// TIA Portal project "Project4_V16" (V16)

(* hardware
DEVICE "S7-1200 station_2"  S7-1200 Station
   slot 0: "Rack_0"  S7-1200 Rack  Rack  V1.0
   slot 1: "PLC_TO_SCADA"  CPU 1214C DC/DC/DC  6ES7 214-1AG40-0XB0  V4.1
DEVICE "S7-1200 station_3"  S7-1200 Station
   slot 0: "Rack_0"  S7-1200 Rack  Rack  V1.0
   slot 1: "PLC_2"  CPU 1214C DC/DC/DC  6ES7 214-1AG40-0XB0  V4.1
DEVICE "S7-1200 station_1"  S7-1200 Station
   slot 0: "Rack_0"  S7-1200 Rack  Rack  V1.0
   slot 1: "PLC_1"  CPU 1212C DC/DC/Rly  6ES7 212-1HE40-0XB0  V4.2
*)

// ===== PLC "PLC_TO_SCADA"  CPU 1214C DC/DC/DC =====

VAR_GLOBAL   // PLC tag table "Default tag table"
   "Tag_1" AT %M0.0 : Bool;
   "Tag_2" AT %M0.1 : Bool;
   "Tag_3" AT %M0.5 : Bool;
   "Tag_4" AT %MD100 : Time;
   "Tag_5" AT %M0.2 : Bool;
   "Tag_6" AT %I0.0 : Bool;
   "Tag_7" AT %I0.1 : Bool;
END_VAR

// folder: System blocks/Program resources

DATA_BLOCK "t0"   // DB1
{ S7_Optimized_Access := 'TRUE' }
AUTHOR : Simatic
FAMILY : IEC
NAME : IEC_TMR
VERSION : 1.0
// stored: InstanceOfName IEC_TIMER
"IEC_TIMER"
BEGIN
END_DATA_BLOCK

// folder: (top level)

ORGANIZATION_BLOCK "Main"   // OB1, LAD, ProgramCycle
TITLE = "Main Program Sweep (Cycle)"
{ S7_Optimized_Access := 'TRUE' }
VERSION : 0.1
   VAR_INPUT
      Initial_Call : Bool;   // Initial call of this OB
      Remanence : Bool;   // =True, if remanent data are available
   END_VAR
BEGIN

REGION Network 1
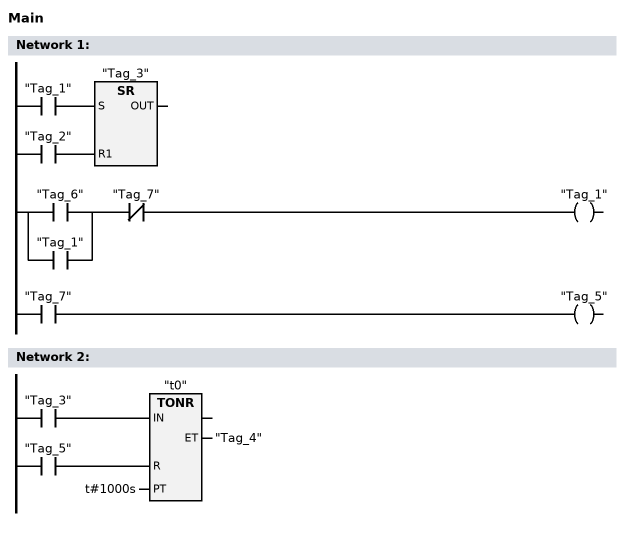
   RUNG wire#powerrail
      Contact( "Tag_1" )
      S_SR(operand := "Tag_3", r1 := wire#w1)
   END_RUNG
   RUNG wire#powerrail
      Contact( "Tag_2" )
   END_RUNG wire#w1
   RUNG wire#powerrail
      Contact( "Tag_6" )
      wire#w2
      I_Contact( "Tag_7" )
      Coil( "Tag_1" )
   END_RUNG
   RUNG wire#powerrail
      Contact( "Tag_1" )
   END_RUNG wire#w2
   RUNG wire#powerrail
      Contact( "Tag_7" )
      Coil( "Tag_5" )
   END_RUNG
   // the same network as SCL:
   IF "Tag_1" THEN
       "Tag_3" := TRUE;   // SR flip-flop
   END_IF;
   IF "Tag_2" THEN "Tag_3" := FALSE; END_IF;
   "Tag_1" := ("Tag_6" OR "Tag_1") AND NOT "Tag_7";
   "Tag_5" := "Tag_7";
END_REGION

REGION Network 2
   "t0".TONR(IN := "Tag_3", R := "Tag_5", PT := t#1000s, ET => "Tag_4");
END_REGION
END_ORGANIZATION_BLOCK

// ===== PLC "PLC_2"  CPU 1214C DC/DC/DC =====

DATA_BLOCK "DB"   // DB1
{ S7_Optimized_Access := 'FALSE' }
VERSION : 0.1
   VAR
      DataReceive : String;
   END_VAR
BEGIN
END_DATA_BLOCK

ORGANIZATION_BLOCK "Main"   // OB1, LAD, ProgramCycle
TITLE = "Main Program Sweep (Cycle)"
{ S7_Optimized_Access := 'TRUE' }
VERSION : 0.1
   VAR_INPUT
      Initial_Call : Bool;   // Initial call of this OB
      Remanence : Bool;   // =True, if remanent data are available
   END_VAR
BEGIN
END_ORGANIZATION_BLOCK

// ===== PLC "PLC_1"  CPU 1212C DC/DC/Rly =====

VAR_GLOBAL   // PLC tag table "Default tag table"
   "Start" AT %I0.0 : Bool;
   "Pause" AT %I0.1 : Bool;
   "Tag_3" AT %M0.0 : Bool;
   "Stop" AT %I0.2 : Bool;
   "Tag_5" AT %MD100 : Time;
END_VAR

DATA_BLOCK "Data_block_1"   // DB1
{ S7_Optimized_Access := 'FALSE' }
VERSION : 0.1
   VAR
      CodeType : Int;
      Data_leng : Int;
      ID_AGV : Int := 0;
      Position : DInt;
      Speed : Int;
      ID_Station : Int;
      Step_Line : Int;
      Status_AGV : Int;
   END_VAR
BEGIN
END_DATA_BLOCK

// folder: System blocks/Program resources

DATA_BLOCK "timerr"   // DB4
{ S7_Optimized_Access := 'TRUE' }
AUTHOR : Simatic
FAMILY : IEC
NAME : IEC_TMR
VERSION : 1.0
// stored: InstanceOfName IEC_TIMER
"IEC_TIMER"
BEGIN
END_DATA_BLOCK

// folder: (top level)

ORGANIZATION_BLOCK "Main"   // OB1, LAD, ProgramCycle
TITLE = "Main Program Sweep (Cycle)"
{ S7_Optimized_Access := 'TRUE' }
VERSION : 0.1
   VAR_INPUT
      Initial_Call : Bool;   // Initial call of this OB
      Remanence : Bool;   // =True, if remanent data are available
   END_VAR
BEGIN

REGION Network 1
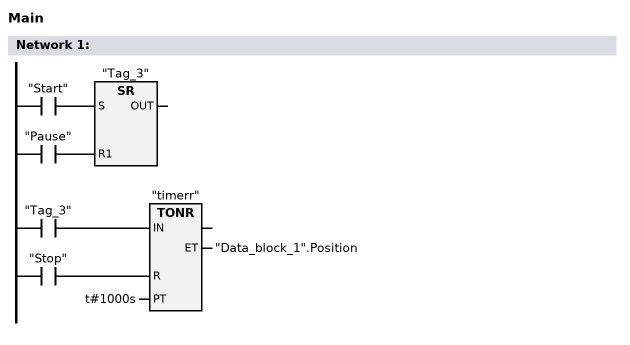
   IF "Start" THEN
       "Tag_3" := TRUE;   // SR flip-flop
   END_IF;
   IF "Pause" THEN "Tag_3" := FALSE; END_IF;
   "timerr".TONR(IN := "Tag_3", R := "Stop", PT := t#1000s, ET => "Data_block_1".Position);
END_REGION
END_ORGANIZATION_BLOCK